ReceiveString_sample_1(
	Prefix:='w' ,
	Suffix:='g' ,
	Timeout:= t#5s,
	Reset:= ,
	ReceivedString:=samplestring_1 ,
	RXbuffer:= RxBuffer1,
	StringReceived=> ,
	Busy=> ,
	Error=> ,
	RxTimeout=> );
ipos_1:=FIND(samplestring_1,'n');

resultWt_1:= MID (samplestring_1,9,ipos_1+1);
Ret_AWt:=STRING_TO_REAL(resultWt_1);


(*==============Ret - B Weight Read==================*)

COMportControl_2(
	Mode:= SERIALLINEMODE_EL6_22B,
	pComIn:= ADR(COMin_2_COMport_2),
	pComOut:= ADR(COMout_2_COMport_2),
	SizeComIn:= SIZEOF(COMin_2_COMport_2),
	TxBuffer:= TxBuffer2,
	RxBuffer:= RxBuffer2,
	Error=> COMportControlError_2,
	ErrorID=> COMportControlErrorID_2);

ReceiveString_sample_2(
	Prefix:='w' ,
	Suffix:='g' ,
	Timeout:= t#5s,
	Reset:= ,
	ReceivedString:=samplestring_2 ,
	RXbuffer:= RxBuffer2,
	StringReceived=> ,
	Busy=> ,
	Error=> ,
	RxTimeout=> );
ipos_1:=FIND(samplestring_2,'n');

resultWt_2:= MID (samplestring_1,9,ipos_2+1);
Ret_BWt:=STRING_TO_REAL(resultWt_2);
END_PROGRAM

(* POU DalaLog, ST *)
PROGRAM DalaLog
VAR

	TON_Indo1: TON;
	TON_Indo2: TON;
	TON_Indo3: TON;
	TON_Indo4: TON;

	TON_Newdaydly: TON;
	TON_NEWDAY: TON;

	TON_NewdaydlyError: TON;

	TON_writedly: TON;

	TON_Opendly: TON;

END_VAR
;
END_PROGRAM

(* POU Initialization, ST *)
PROGRAM Initialization
VAR




END_VAR
;
END_PROGRAM

(* POU Alarms/Piston_Alarms, ST *)
PROGRAM Piston_Alarms
VAR
	TON_ConeFeedingPistonOff: BOOL;
	F_TRIG_ConeFeedingPiston: F_TRIG;
	bAConeFeedingPistonOff: BOOL;
	RS_ErrorConeFeedPistonHome: Rs_Error;
	RS_ErrorConeFeedPistonEnd: Rs_Error;
	HMIFeedPistonHome: STRING;
	HMIFeedPistonEnd: STRING;
	HMIFeedPiston: STRING;

	TON_ConeForwardPistonOff: BOOL;
	F_TRIG_ConeForwardPiston: F_TRIG;
	bAConeForwardPistonOff: BOOL;
	RS_ErrorConeForwardPistonHome: Rs_Error;
	RS_ErrorConeForwardPistonEnd: Rs_Error;
	HMIForwardPistonHome: STRING;
	HMIForwardPistonEnd: STRING;
	HMIForwardPiston: STRING;

	TON_ConeReversePistonOff: BOOL;
	F_TRIG_ConeReversePiston: F_TRIG;
	bAConeReversePistonOff: BOOL;
	RS_ErrorConeReversePistonHome: Rs_Error;
	RS_ErrorConeReversePistonEnd: Rs_Error;
	HMIReversePistonHome: STRING;
	HMIReversePistonEnd: STRING;
	HMIReversePiston: STRING;

	TON_ConeTiltingPistonOff: BOOL;
	F_TRIG_ConeTiltingPiston: F_TRIG;
	bAConeTiltingPistonOff: BOOL;
	RS_ErrorConeTiltingPistonHome: Rs_Error;
	RS_ErrorConeTiltingPistonEnd: Rs_Error;
	HMITiltingPistonHome: STRING;
	HMITiltingPistonEnd: STRING;
	HMITiltingPiston: STRING;
	bATiltingPisHomeRsError: BOOL;
	bATiltingPisEndRsError: BOOL;

	TON_Wrapping1PistonOff: BOOL;
	F_TRIG_Wrapping1Piston: F_TRIG;
	bAWrapping1PistonOff: BOOL;
	RS_ErrorWrapping1PistonHome: Rs_Error;
	RS_ErrorWrapping1PistonEnd: Rs_Error;
	HMIWrapping1PistonHome: STRING;
	HMIWrapping1PistonEnd: STRING;
	HMIWrapping1Piston: STRING;
	bAWrapping1PisHomeRsError: BOOL;
	bAWrapping1PisEndRsError: BOOL;

	TON_Wrapping2PistonOff: BOOL;
	F_TRIG_Wrapping2Piston: F_TRIG;
	bAWrapping2PistonOff: BOOL;
	RS_ErrorWrapping2PistonHome: Rs_Error;
	RS_ErrorWrapping2PistonEnd: Rs_Error;
	HMIWrapping2PistonHome: STRING;
	HMIWrapping2PistonEnd: STRING;
	HMIWrapping2Piston: STRING;
	bAWrapping2PisHomeRsError: BOOL;
	bAWrapping2PisEndRsError: BOOL;
END_VAR
(*......................................Cone Feeding Piston Home Alarm.............................*)

F_TRIG_ConeFeedingPiston(CLK:=bQAConeFeedPisOn , Q=> );

IF F_TRIG_ConeFeedingPiston.Q THEN bAConeFeedingPistonOff:=TRUE;END_IF
IF bIConeFeedingPistonHome THEN bAConeFeedingPistonOff:=FALSE;END_IF



RS_ErrorConeFeedPistonHome(
	bValveOutOn:= bAConeFeedingPistonOff,
	bReedSwithIn:=  bIConeFeedingPistonHome ,
	bErroReset:= bErrorReset ,
	sMsgIn:= ,
	RS_ErrChkDly:=t#5s ,
	bRsError=>bAConeFeedingPistonHomeRsError ,
	sMsgOut=> );

IF RS_ErrorConeFeedPistonHome.bRsError THEN
RS_ErrorConeFeedPistonHome.sMsgIn:='Cone Feeding Piston Home Sensor Timeout Error' ;
ELSE
RS_ErrorConeFeedPistonHome.sMsgIn:='Continue Machine Operation' ;
END_IF
HMIFeedPistonHome:=RS_ErrorConeFeedPistonHome.sMsgIn;

IF bAConeFeedingPistonHomeRsError THEN HMIFeedPiston:=HMIFeedPistonHome;
ELSIF bAConeFeedingPistonEndRsError THEN  HMIFeedPiston:=HMIFeedPistonEnd;
ELSIF NOT bAConeFeedingPistonHomeRsError AND NOT bAConeFeedingPistonEndRsError THEN
HMIFeedPiston:='Continue Machine Running';END_IF


(*......................................Cone Feeding Piston Alarm.............................*)


RS_ErrorConeFeedPistonEnd(
	bValveOutOn:= bQAConeFeedPisOn,
	bReedSwithIn:=  bIConeFeedingPistonEnd ,
	bErroReset:= bErrorReset ,
	sMsgIn:= ,
	RS_ErrChkDly:=t#10s ,
	bRsError=>bAConeFeedingPistonEndRsError ,
	sMsgOut=> );

IF RS_ErrorConeFeedPistonEnd.bRsError THEN
RS_ErrorConeFeedPistonEnd.sMsgIn:='Cone Feeding Piston End Sensor Timeout Error' ;
ELSE
RS_ErrorConeFeedPistonEnd.sMsgIn:='Continue Machine Operation' ;
END_IF
HMIFeedPistonEnd:=RS_ErrorConeFeedPistonEnd.sMsgIn;


(*......................................Cone Forward Piston Home Alarm.............................*)

F_TRIG_ConeForwardPiston(CLK:=bQAForwardPistonOn , Q=> );

IF F_TRIG_ConeForwardPiston.Q THEN bAConeForwardPistonOff:=TRUE;END_IF
IF bIForwardPistonHome THEN bAConeForwardPistonOff:=FALSE;END_IF



RS_ErrorConeForwardPistonHome(
	bValveOutOn:= bAConeForwardPistonOff,
	bReedSwithIn:=  bIForwardPistonHome ,
	bErroReset:= bErrorReset ,
	sMsgIn:= ,
	RS_ErrChkDly:=t#5s ,
	bRsError=>bAForwardPisHomeRsError ,
	sMsgOut=> );

IF RS_ErrorConeForwardPistonHome.bRsError THEN
RS_ErrorConeForwardPistonHome.sMsgIn:='Cone Forward Piston Home Sensor Timeout Error' ;
ELSE
RS_ErrorConeForwardPistonHome.sMsgIn:='Continue Machine Operation' ;
END_IF
HMIForwardPistonHome:=RS_ErrorConeForwardPistonHome.sMsgIn;

IF bAForwardPisHomeRsError THEN HMIForwardPiston:=HMIForwardPistonHome;
ELSIF bAForwardPisEndRsError THEN  HMIForwardPiston:=HMIForwardPistonEnd;
ELSIF NOT bAForwardPisHomeRsError AND NOT bAForwardPisEndRsError THEN
HMIForwardPiston:='Continue Machine Running';END_IF


(*......................................Cone Forward Piston End Alarm.............................*)


RS_ErrorConeForwardPistonEnd(
	bValveOutOn:= bQAForwardPistonOn,
	bReedSwithIn:=  bIForwardPistonEnd ,
	bErroReset:= bErrorReset ,
	sMsgIn:= ,
	RS_ErrChkDly:=t#10s ,
	bRsError=>bAForwardPisEndRsError ,
	sMsgOut=> );

IF RS_ErrorConeForwardPistonEnd.bRsError THEN
RS_ErrorConeForwardPistonEnd.sMsgIn:='Cone Forward Piston End Sensor Timeout Error' ;
ELSE
RS_ErrorConeForwardPistonEnd.sMsgIn:='Continue Machine Operation' ;
END_IF
HMIForwardPistonEnd:=RS_ErrorConeForwardPistonEnd.sMsgIn;


(*......................................Cone Reverse Piston Home Alarm.............................*)

F_TRIG_ConeReversePiston(CLK:=bQAReversePistonOn , Q=> );

IF F_TRIG_ConeReversePiston.Q THEN bAConeReversePistonOff:=TRUE;END_IF
IF bIReversePistonHome THEN bAConeReversePistonOff:=FALSE;END_IF



RS_ErrorConeReversePistonHome(
	bValveOutOn:= bAConeReversePistonOff,
	bReedSwithIn:=  bIReversePistonHome ,
	bErroReset:= bErrorReset ,
	sMsgIn:= ,
	RS_ErrChkDly:=t#5s ,
	bRsError=>bAReversePisHomeRsError ,
	sMsgOut=> );

IF RS_ErrorConeReversePistonHome.bRsError THEN
RS_ErrorConeReversePistonHome.sMsgIn:='Cone Reverse Piston Home Sensor Timeout Error' ;
ELSE
RS_ErrorConeReversePistonHome.sMsgIn:='Continue Machine Operation' ;
END_IF
HMIReversePistonHome:=RS_ErrorConeReversePistonHome.sMsgIn;

IF bAReversePisHomeRsError THEN HMIReversePiston:=HMIReversePistonHome;
ELSIF bAReversePisEndRsError THEN  HMIReversePiston:=HMIReversePistonEnd;
ELSIF NOT bAReversePisHomeRsError AND NOT bAReversePisEndRsError THEN
HMIReversePiston:='Continue Machine Running';END_IF


(*......................................Cone Reverse Piston End Alarm.............................*)


RS_ErrorConeReversePistonEnd(
	bValveOutOn:= bQAReversePistonOn,
	bReedSwithIn:=  bIReversePistonEnd ,
	bErroReset:= bErrorReset ,
	sMsgIn:= ,
	RS_ErrChkDly:=t#10s ,
	bRsError=>bAReversePisEndRsError ,
	sMsgOut=> );

IF RS_ErrorConeReversePistonEnd.bRsError THEN
RS_ErrorConeReversePistonEnd.sMsgIn:='Cone Reverse Piston End Sensor Timeout Error' ;
ELSE
RS_ErrorConeReversePistonEnd.sMsgIn:='Continue Machine Operation' ;
END_IF
HMIReversePistonEnd:=RS_ErrorConeReversePistonEnd.sMsgIn;




(*......................................Cone Tilting Piston Home Alarm.............................*)

F_TRIG_ConeTiltingPiston(CLK:=bQAReversePistonOn , Q=> );

IF F_TRIG_ConeTiltingPiston.Q THEN bAConeTiltingPistonOff:=TRUE;END_IF
IF bIReversePistonHome THEN bAConeTiltingPistonOff:=FALSE;END_IF



RS_ErrorConeTiltingPistonHome(
	bValveOutOn:= bAConeReversePistonOff,
	bReedSwithIn:=  bIReversePistonHome ,
	bErroReset:= bErrorReset ,
	sMsgIn:= ,
	RS_ErrChkDly:=t#5s ,
	bRsError=>bATiltingPisHomeRsError ,
	sMsgOut=> );

IF RS_ErrorConeTiltingPistonHome.bRsError THEN
RS_ErrorConeTiltingPistonHome.sMsgIn:='Cone Tilting Piston Home Sensor Timeout Error' ;
ELSE
RS_ErrorConeTiltingPistonHome.sMsgIn:='Continue Machine Operation' ;
END_IF
HMITiltingPistonHome:=RS_ErrorConeTiltingPistonHome.sMsgIn;

IF bATiltingPisHomeRsError THEN HMITiltingPiston:=HMITiltingPistonHome;
ELSIF bATiltingPisEndRsError THEN  HMITiltingPiston:=HMITiltingPistonEnd;
ELSIF NOT bATiltingPisHomeRsError AND NOT bATiltingPisEndRsError THEN
HMITiltingPiston:='Continue Machine Running';END_IF


(*......................................Cone Tilting Piston End Alarm.............................*)


RS_ErrorConeTiltingPistonEnd(
	bValveOutOn:= bQAReversePistonOn,
	bReedSwithIn:=  bIReversePistonEnd ,
	bErroReset:= bErrorReset ,
	sMsgIn:= ,
	RS_ErrChkDly:=t#10s ,
	bRsError=>bATiltingPisEndRsError ,
	sMsgOut=> );

IF RS_ErrorConeTiltingPistonEnd.bRsError THEN
RS_ErrorConeTiltingPistonEnd.sMsgIn:='Cone Tilting Piston End Sensor Timeout Error' ;
ELSE
RS_ErrorConeTiltingPistonEnd.sMsgIn:='Continue Machine Operation' ;
END_IF
HMITiltingPistonEnd:=RS_ErrorConeTiltingPistonEnd.sMsgIn;




(*......................................Wrapping1 Piston Home Alarm.............................*)

F_TRIG_Wrapping1Piston(CLK:=bQAReversePistonOn , Q=> );

IF F_TRIG_Wrapping1Piston.Q THEN bAWrapping1PistonOff:=TRUE;END_IF
IF bIReversePistonHome THEN bAWrapping1PistonOff:=FALSE;END_IF



RS_ErrorWrapping1PistonHome(
	bValveOutOn:= bAConeReversePistonOff,
	bReedSwithIn:=  bIReversePistonHome ,
	bErroReset:= bErrorReset ,
	sMsgIn:= ,
	RS_ErrChkDly:=t#5s ,
	bRsError=>bAWrapping1PisHomeRsError ,
	sMsgOut=> );

IF RS_ErrorWrapping1PistonHome.bRsError THEN
RS_ErrorWrapping1PistonHome.sMsgIn:='Cone Wrapping1 Piston Home Sensor Timeout Error' ;
ELSE
RS_ErrorWrapping1PistonHome.sMsgIn:='Continue Machine Operation' ;
END_IF
HMIWrapping1PistonHome:=RS_ErrorWrapping1PistonHome.sMsgIn;

IF bAWrapping1PisHomeRsError THEN HMIWrapping1Piston:=HMIWrapping1PistonHome;
ELSIF bAWrapping1PisEndRsError THEN  HMIWrapping1Piston:=HMIWrapping1PistonEnd;
ELSIF NOT bAWrapping1PisHomeRsError AND NOT bAWrapping1PisEndRsError THEN
HMIWrapping1Piston:='Continue Machine Running';END_IF


(*......................................Cone Wrapping1 Piston End Alarm.............................*)


RS_ErrorWrapping1PistonEnd(
	bValveOutOn:= bQAReversePistonOn,
	bReedSwithIn:=  bIReversePistonEnd ,
	bErroReset:= bErrorReset ,
	sMsgIn:= ,
	RS_ErrChkDly:=t#10s ,
	bRsError=>bAWrapping1PisEndRsError ,
	sMsgOut=> );

IF RS_ErrorWrapping1PistonEnd.bRsError THEN
RS_ErrorWrapping1PistonEnd.sMsgIn:='Cone Wrapping1 Piston End Sensor Timeout Error' ;
ELSE
RS_ErrorWrapping1PistonEnd.sMsgIn:='Continue Machine Operation' ;
END_IF
HMIWrapping1PistonEnd:=RS_ErrorWrapping1PistonEnd.sMsgIn;




(*......................................Wrapping2 Piston Home Alarm.............................*)

F_TRIG_Wrapping2Piston(CLK:=bQAReversePistonOn , Q=> );

IF F_TRIG_Wrapping2Piston.Q THEN bAWrapping2PistonOff:=TRUE;END_IF
IF bIReversePistonHome THEN bAWrapping2PistonOff:=FALSE;END_IF



RS_ErrorWrapping2PistonHome(
	bValveOutOn:= bAConeReversePistonOff,
	bReedSwithIn:=  bIReversePistonHome ,
	bErroReset:= bErrorReset ,
	sMsgIn:= ,
	RS_ErrChkDly:=t#5s ,
	bRsError=>bAWrapping2PisHomeRsError ,
	sMsgOut=> );

IF RS_ErrorWrapping2PistonHome.bRsError THEN
RS_ErrorWrapping2PistonHome.sMsgIn:='Cone Wrapping2 Piston Home Sensor Timeout Error' ;
ELSE
RS_ErrorWrapping2PistonHome.sMsgIn:='Continue Machine Operation' ;
END_IF
HMIWrapping2PistonHome:=RS_ErrorWrapping2PistonHome.sMsgIn;

IF bAWrapping2PisHomeRsError THEN HMIWrapping2Piston:=HMIWrapping2PistonHome;
ELSIF bAWrapping2PisEndRsError THEN  HMIWrapping2Piston:=HMIWrapping2PistonEnd;
ELSIF NOT bAWrapping2PisHomeRsError AND NOT bAWrapping2PisEndRsError THEN
HMIWrapping2Piston:='Continue Machine Running';END_IF


(*......................................Cone Wrapping2 Piston End Alarm.............................*)


RS_ErrorWrapping2PistonEnd(
	bValveOutOn:= bQAReversePistonOn,
	bReedSwithIn:=  bIReversePistonEnd ,
	bErroReset:= bErrorReset ,
	sMsgIn:= ,
	RS_ErrChkDly:=t#10s ,
	bRsError=>bAWrapping2PisEndRsError ,
	sMsgOut=> );

IF RS_ErrorWrapping2PistonEnd.bRsError THEN
RS_ErrorWrapping2PistonEnd.sMsgIn:='Cone Wrapping2 Piston End Sensor Timeout Error' ;
ELSE
RS_ErrorWrapping2PistonEnd.sMsgIn:='Continue Machine Operation' ;
END_IF
HMIWrapping2PistonEnd:=RS_ErrorWrapping2PistonEnd.sMsgIn;
END_PROGRAM

(* POU Rs_Error, ST *)
FUNCTION_BLOCK Rs_Error
VAR_INPUT
	bValveOutOn: BOOL;
	bReedSwithIn: BOOL;
	bErroReset: BOOL;
	sMsgIn: STRING;
	RS_ErrChkDly: TIME;
END_VAR
VAR_OUTPUT
	bRsError: BOOL;
	sMsgOut: STRING;
END_VAR
VAR
	FbStep: INT;
	Timer1: TON;
END_VAR
CASE FbStep OF


	0:	Timer1(IN:=FALSE); FbStep:=FbStep+1;

	1:	IF bValveOutOn THEN FbStep:=FbStep+1; END_IF

	2:	Timer1(IN:=TRUE , PT:=RS_ErrChkDly , Q=> , ET=> );
		IF Timer1.Q THEN FbStep:=FbStep+1;
		ELSIF NOT  Timer1.Q AND bReedSwithIn THEN  FbStep:=0; END_IF

	3:	IF bReedSwithIn THEN  FbStep:=FbStep+1;
		ELSIF NOT bReedSwithIn THEN FbStep:=FbStep+2; END_IF

	4:	IF  NOT bValveOutOn THEN sMsgOut:=sMsgIn;  FbStep:=0; END_IF

	5:	bRsError:=TRUE; FbStep:=FbStep+1;

	6:	IF   bReedSwithIn AND   bErroReset THEN bRsError:=FALSE; sMsgOut:='' ;  FbStep:=0;
		ELSIF   NOT bReedSwithIn AND   bRsError  AND  bErroReset THEN bRsError:=FALSE;   sMsgOut:='' ;   FbStep:=0;
		 END_IF

END_CASE
END_FUNCTION_BLOCK

(* POU Piston_Errors, ST *)
PROGRAM Piston_Errors
VAR
END_VAR
;
END_PROGRAM

(* POU TowerLamp, ST *)
PROGRAM TowerLamp
VAR
	bQTLRed: BOOL;
	bQATLRed: BOOL;
	bAIntBlinkAuto: BOOL;
	bQBuzzer: BOOL;
	bQABuzzer: BOOL;
	bQTLGreen: BOOL;
	bQATLGreen: BOOL;
	bQATLGreenBlnkAuto: BOOL;
	bQTLAmber: BOOL;
	bQATLAmber: BOOL;
	bAEmergencyPressed: BOOL;
	BlinkTimer_1: TON;
	ERROR_ALERT: BOOL;
	BlinkTimer_2: TON;
	BlinkTimer3: TON;
	BlinkTimer4: TON;
	bQAGreenBlnkAuto: BOOL;
	BlinkTimer5: TON;
	BlinkTimer6: TON;
	bTLBlinkOn: BOOL;
	BlinkTimer1: TON;
	BlinkTimer2: TON;
END_VAR
IF bAutoModeOn
THEN
bQTLRed:=  bQATLRed OR bAIntBlinkAuto;

		bQBuzzer:= bQABuzzer;

		bQTLGreen :=(bQATLGreen OR bAIntBlinkAuto OR bQATLGreenBlnkAuto);

		bQTLAmber:=bQATLAmber OR bAIntBlinkAuto;

IF bIMcStopPb OR Stop_TapHmi
THEN bAEmergencyPressed:=TRUE;
ELSE bAEmergencyPressed:=FALSE;
END_IF


BlinkTimer_1(IN:=(ERROR_ALERT AND NOT BlinkTimer_2.Q) , PT:= t#0.5s, Q=> , ET=> );

BlinkTimer_2(IN:= BlinkTimer_1.Q, PT:=t#1.3s , Q=> , ET=> );


BlinkTimer3(IN:= (bAEmergencyPressed AND NOT BlinkTimer4.Q) , PT:= t#0.5s, Q=> , ET=> );

BlinkTimer4(IN:= BlinkTimer3.Q, PT:=t#1.3s , Q=> , ET=> );




IF bAutoModeOn AND (ERROR_ALERT OR bPauseSeq)  AND NOT  bAEmergencyPressed THEN
 bQATLAmber:=TRUE; bQATLGreen:=FALSE;bQATLRed:=FALSE;  ELSE bQATLAmber:=FALSE;
END_IF

IF bAutoModeOn AND (BlinkTimer_1.Q OR BlinkTimer3.Q)
THEN  bQABuzzer:=TRUE;
ELSE bQABuzzer:=FALSE;
END_IF


IF bAutoModeOn AND bAEmergencyPressed
 THEN bQATLRed:=TRUE;bQATLGreen:=FALSE;bQATLAmber:=FALSE;
END_IF

IF bAutoModeOn AND NOT  bAEmergencyPressed AND NOT ERROR_ALERT AND
bMCStartInAuto AND NOT bAMainIntStarted AND NOT IntAllOver  AND NOT  bPauseSeq THEN
bQAGreenBlnkAuto:=TRUE;bQATLAmber:=FALSE;bQATLRed:=FALSE;
ELSE bQAGreenBlnkAuto:=FALSE;
END_IF



BlinkTimer5(IN:= (bQAGreenBlnkAuto AND NOT BlinkTimer6.Q) , PT:= t#0.5s, Q=> , ET=> );
BlinkTimer6(IN:= BlinkTimer5.Q, PT:=t#1.3s , Q=> , ET=> );

IF bAutoModeOn AND BlinkTimer5.Q
THEN bQATLGreenBlnkAuto:=TRUE;
ELSE bQATLGreenBlnkAuto:=FALSE;
END_IF


IF bAutoModeOn AND bMcStartInAuto AND bAMainIntStarted AND NOT  bPauseSeq
AND NOT ERROR_ALERT  AND NOT  bAEmergencyPressed THEN
bTLBlinkOn:=TRUE; bQATLGreen:=FALSE;bQATLAmber:=FALSE; bQATLRed:=FALSE;
ELSE  bTLBlinkOn:=FALSE;
 END_IF

BlinkTimer1(IN:=(bTLBlinkOn AND NOT BlinkTimer2.Q) , PT:= t#0.5s, Q=> , ET=> );

BlinkTimer2(IN:= BlinkTimer1.Q, PT:=t#1.3s , Q=> , ET=> );

IF bAutoModeOn AND  BlinkTimer1.Q
THEN bAIntBlinkAuto:=TRUE;
 ELSE  bAIntBlinkAuto:=FALSE;
 END_IF


IF  bAutoModeOn AND bMCStartInAuto  AND NOT  bAEmergencyPressed AND NOT  bPauseSeq
AND NOT ERROR_ALERT AND NOT bAMainIntStarted AND IntAllOver THEN
 bQATLGreen :=TRUE;bQATLAmber:=FALSE; bQATLRed:=FALSE;
ELSIF NOT IntAllOver THEN bQATLGreen:=FALSE;
 END_IF

END_IF




IF NOT bIAutoManualSwitch
THEN bQATLAmber:=FALSE;bQATLRed:=FALSE;bQATLGreen:=FALSE;bQABuzzer:=FALSE;bAIntBlinkAuto:=FALSE;
END_IF


IF NOT bIAutoManualSwitch THEN bQTLRed:=FALSE;bQBuzzer:=FALSE;bQTLGreen:=FALSE;
bQTLAmber:=FALSE;bQATLRed:=FALSE;bQABuzzer:=FALSE;bQATLGreen:=FALSE;
bQATLGreenBlnkAuto:=FALSE;bQATLAmber:=FALSE;
bAIntBlinkAuto:=FALSE;END_IF
END_PROGRAM

(* Visualisation Auto
1 more shapes without text or variables
*)
